(* IEC 61131-3 sources: _TiaPortal14/TEST_SCL_Schleifmaschine/Schleifmaschine/net5.0-windows/ConfigTests/Schleifmaschine_1, 1 file *)

(* ---- testProgramm.st ---- *)
FUNCTION_BLOCK TestProgramm
VAR_INPUT
END_VAR
VAR_OUTPUT
END_VAR
VAR
    ZyklusAktiv: BOOL;
	Zeit: TON;
END_VAR

(*  *********************************************************** *)
(*  Schleifmaschine mit zwei Drehzahlen                         *)
(*  *********************************************************** *)
